// TIA Portal V21 export
FUNCTION "DiFc" : Void   // FC101, LAD
TITLE = DIFC
{ S7_Optimized_Access := 'TRUE' }
// stored: AutoNumber false, SetENOAutomatically false
BEGIN

REGION Network 1 (SCL): DI Final
   "DiFinal".ControlKey := "DiSimulation".ControlKey OR "ControlKey";
   "DiFinal".EmergencyStop := "DiSimulation".EmergencyStop OR "EmergencyStop";
   "DiFinal".CompressedAirPressureLow := "DiSimulation".CompressedAirPressureLow OR "CompressedAirPressureLow";
   "DiFinal".PowerFailure := "DiSimulation".PowerFailure OR "PowerFailure";
   "DiFinal".PowerReset := "DiSimulation".PowerReset OR "PowerReset";
   "DiFinal".MagneticMixerFeedback := "DiSimulation".MagneticMixerFeedback OR "MagneticMixerFeedback";
   "DiFinal".CipPumpFeedback := "DiSimulation".CipPumpFeedback OR "CipPumpFeedback";
   "DiFinal".MagneticMixerOverload := "DiSimulation".MagneticMixerOverload OR "MagneticMixerOverload";
   "DiFinal".CipPumpOverload := "DiSimulation".CipPumpOverload OR "CipPumpOverload";
   "DiFinal".RuptureDisc := "DiSimulation".RuptureDisc OR "RuptureDisc";
   "DiFinal".Cp01FlowSwitch := "DiSimulation".Cp01FlowSwitch OR "Cp01FlowSwitch";
   "DiFinal".DiSpare1 := "DiSimulation".DiSpare1 OR "DiSpare1";
   "DiFinal".DiSpare2 := "DiSimulation".DiSpare2 OR "DiSpare2";
   "DiFinal".MMHighSpeedSensor := "DiSimulation".MMHighSpeedSensor OR "MMHighSpeedSensor";
   "DiFinal".DiSpare3 := "DiSimulation".DiSpare3 OR "DiSpare3";
   "DiFinal".DiSpare4 := "DiSimulation".DiSpare4 OR "DiSpare4";
   "DiFinal".DiSpare5 := "DiSimulation".DiSpare5 OR "DiSpare5";
   "DiFinal".DiSpare6 := "DiSimulation".DiSpare6 OR "DiSpare6";
   "DiFinal".DiSpare7 := "DiSimulation".DiSpare7 OR "DiSpare7";
   "DiFinal".DiSpare8 := "DiSimulation".DiSpare8 OR "DiSpare8";
   "DiFinal".DiSpare9:= "DiSimulation".DiSpare9 OR "DiSpare9";
   "DiFinal".DiSpare10 := "DiSimulation".DiSpare10 OR "DiSpare10";
END_REGION
END_FUNCTION
